// TIA Portal V20 export
DATA_BLOCK "BK19"   // DB266
// stored: MemoryReserve 100
   VAR
      "X10-1 SPARE" : Bool;
      "X10-2 SPARE" : Bool;
      "X12-1 SPARE" : Bool;
      "X12-2 SPARE" : Bool;
      "X14-1 WEIGHT DETECT SENSOR" : Bool;
      "X14-2 SPARE" : Bool;
      "X16-1 MAIN VALVE DIGITAL PRESSURE SWITCH OUT1" : Bool;
      "X16-2 MAIN VALVE DIGITAL PRESSURE SWITCH OUT2" : Bool;
   END_VAR
BEGIN
END_DATA_BLOCK
